{attribute 'GeneratedUsingTerminal: EL5101-0011-0016'}
{attribute addProperty BoxType "EL5101-0011-0016"}
{attribute addProperty Id "ControlAT %Q*Control_BD9A418F1Set_counter_valueAT %Q*UDINT4"}
{attribute addProperty CRC "350482255"}
{attribute addProperty Size "5"}
TYPE ENC_Control_14E3EF4F :
STRUCT
	{attribute addProperty Name "Control"}
	Control AT %Q* : Control_BD9A418F;
	{attribute addProperty Name "Set_counter_value"}
	Set_counter_value AT %Q* : UDINT;
END_STRUCT
END_TYPE

(* stored: Version 1.2.0.0, ProductVersion 3.1.4024.9
   DUT ENC_Control_14E3EF4F: Id {591be189-ecf0-48c9-8cf3-7d624b7a3305} *)
